TYPE ST_SCANNER_HostAck :
STRUCT
	bSetHostAckTimeOut				: BOOL;
	tAckTimeOut						: TIME;
	bGoodReadResponse				: BOOL;
	bBadReadResponse				: BOOL;
END_STRUCT
END_TYPE

(* stored: Version 1.1.0.1, ProductVersion 3.1.4024.15
   DUT ST_SCANNER_HostAck: Id {fca606a5-7eef-4142-b24f-43404294aee8} *)
